PROGRAM PrgMqttCom_Blinds_Publisher
VAR
	fbMqttClient : FB_IotMqttClient;
	bSetParameter : BOOL := TRUE;
	bConnect : BOOL := TRUE;
	
	(* published message *)
	sTopicSelectRoom : STRING(255);//:= 'Staff Room';
	sTopicSelectBulkCommand : STRING(255) := 'Blind Selection';
	//sTopicSelectBoardroom : STRING(255) := 'Boardroom';
	
	bSelectStaffRoom : BOOL;
	bSelectCommunalArea : BOOL;
	bSelectBoardroom : BOOL;
	
	sPayloadCommand : STRING(255);// := 'Up';
//	sPayloadCommandDown : STRING(255) := 'Down';
//	sPayloadCommandStop : STRING(255) := 'Stop';
//	sPayloadCommandTilt : STRING(255) := 'Tilt';

	bCommandUp : BOOL;
	bCommandDown : BOOL;
	bCommandStop : BOOL;
	bCommandTilt : BOOL;
	
	bulkCommandPackage :STRING;
	
	i: INT;
	fbTimer : TON := (PT:=T#1S);
	fbTimerTilt : TON := (PT:=T#0.5S);
	
	fbMessageQueue : FB_IotMqttMessageQueue;
	fbMessage : FB_IotMqttMessage;
	
	hrErrorOccurred : HRESULT; // contains the latest occurred error
END_VAR

IF bSetParameter THEN
	bSetParameter := FALSE;
	fbMqttClient.sHostName:= '10.199.143.2';
	fbMqttClient.nHostPort:= 1883;
	fbMqttClient.sClientId:= 'CX2040_Blinds'; 
	fbMqttClient.sTopicPrefix:= ''; 
	fbMqttClient.nKeepAlive:= 60; 
//	fbMqttClient.sUserName:= ;
//	fbMqttClient.sUserPassword:= ; 
//	fbMqttClient.stWill:= ; 
//	fbMqttClient.stTLS:= ;
	fbMqttClient.ipMessageQueue := fbMessageQueue;
END_IF

fbMqttClient.Execute(bConnect);
IF fbMqttClient.bError THEN
	// add your error logging here
	hrErrorOccurred := fbMqttClient.hrErrorCode;
END_IF

IF bSelectStaffRoom THEN
	bSelectStaffRoom := FALSE;
	sTopicSelectRoom := 'Staff Room';
	bulkCommandPackage := fConvertBoolArrayToString(boolArray := BackgroundComms.BlindCommandTable[0].SelectBlindsBulkCommand);
END_IF

IF bSelectCommunalArea THEN
	bSelectCommunalArea := FALSE;
	sTopicSelectRoom := 'Communal Area';
	bulkCommandPackage := fConvertBoolArrayToString(boolArray := BackgroundComms.BlindCommandTable[1].SelectBlindsBulkCommand);
END_IF

IF bSelectBoardroom THEN
	bSelectBoardroom := FALSE;
	sTopicSelectRoom := 'Boardroom';
	bulkCommandPackage := fConvertBoolArrayToString(boolArray := BackgroundComms.BlindCommandTable[2].SelectBlindsBulkCommand);
END_IF



IF bCommandUp THEN
	bCommandUp := FALSE;
	sPayloadCommand := 'Up';
	IF sTopicSelectRoom = 'Staff Room' THEN
		bSelectStaffRoom := TRUE;
	ELSIF sTopicSelectRoom = 'Communal Area' THEN
		bulkCommandPackage := fConvertBoolArrayToString(boolArray := BackgroundComms.BlindCommandTable[1].SelectBlindsBulkCommand);
	ELSIF sTopicSelectRoom = 'Boardroom' THEN
		bulkCommandPackage := fConvertBoolArrayToString(boolArray := BackgroundComms.BlindCommandTable[2].SelectBlindsBulkCommand);
	END_IF
END_IF

IF bCommandDown THEN
	bCommandDown := FALSE;
	sPayloadCommand := 'Down';
	IF sTopicSelectRoom = 'Staff Room' THEN
		bSelectStaffRoom := TRUE;//bulkCommandPackage := fConvertBoolArrayToString(boolArray := BackgroundComms.BlindCommandTable[0].SelectBlindsBulkCommand);
	ELSIF sTopicSelectRoom = 'Communal Area' THEN
		bulkCommandPackage := fConvertBoolArrayToString(boolArray := BackgroundComms.BlindCommandTable[1].SelectBlindsBulkCommand);
	ELSIF sTopicSelectRoom = 'Boardroom' THEN
		bulkCommandPackage := fConvertBoolArrayToString(boolArray := BackgroundComms.BlindCommandTable[2].SelectBlindsBulkCommand);
	END_IF
END_IF

IF bCommandStop THEN
	bCommandStop := FALSE;
	sPayloadCommand := 'Stop';
	IF sTopicSelectRoom = 'Staff Room' THEN
		bSelectStaffRoom := TRUE;//bulkCommandPackage := fConvertBoolArrayToString(boolArray := BackgroundComms.BlindCommandTable[0].SelectBlindsBulkCommand);
	ELSIF sTopicSelectRoom = 'Communal Area' THEN
		bulkCommandPackage := fConvertBoolArrayToString(boolArray := BackgroundComms.BlindCommandTable[1].SelectBlindsBulkCommand);
	ELSIF sTopicSelectRoom = 'Boardroom' THEN
		bulkCommandPackage := fConvertBoolArrayToString(boolArray := BackgroundComms.BlindCommandTable[2].SelectBlindsBulkCommand);
	END_IF
END_IF

IF bCommandTilt THEN
	bCommandTilt := FALSE;
	sPayloadCommand := 'Tilt';
	IF sTopicSelectRoom = 'Staff Room' THEN
		bSelectStaffRoom := TRUE;//bulkCommandPackage := fConvertBoolArrayToString(boolArray := BackgroundComms.BlindCommandTable[0].SelectBlindsBulkCommand);
	ELSIF sTopicSelectRoom = 'Communal Area' THEN
		bulkCommandPackage := fConvertBoolArrayToString(boolArray := BackgroundComms.BlindCommandTable[1].SelectBlindsBulkCommand);
	ELSIF sTopicSelectRoom = 'Boardroom' THEN
		bulkCommandPackage := fConvertBoolArrayToString(boolArray := BackgroundComms.BlindCommandTable[2].SelectBlindsBulkCommand);
	END_IF
END_IF





IF fbMqttClient.bConnected THEN
	IF sPayloadCommand = 'Tilt' THEN
		fbTimerTilt(IN:=TRUE);
		fbMqttClient.Publish(	sTopic:= sTopicSelectBulkCommand, 
									pPayload:= ADR(bulkCommandPackage), nPayloadSize:= LEN2(ADR(bulkCommandPackage))+1, 
									eQoS:= TcIotMqttQos.AtMostOnceDelivery, bRetain:= FALSE, bQueue:= FALSE );
		fbMqttClient.Publish(	sTopic:= sTopicSelectRoom, 
									pPayload:= ADR(sPayloadCommand), nPayloadSize:= LEN2(ADR(sPayloadCommand))+1, 
									eQoS:= TcIotMqttQos.AtMostOnceDelivery, bRetain:= FALSE, bQueue:= FALSE );
		
		IF fbTimerTilt.Q THEN // publish new payload every second
			sPayloadCommand := 'Stop';
			fbTimerTilt(IN:=FALSE);
			fbMqttClient.Publish(	sTopic:= sTopicSelectBulkCommand, 
									pPayload:= ADR(bulkCommandPackage), nPayloadSize:= LEN2(ADR(bulkCommandPackage))+1, 
									eQoS:= TcIotMqttQos.AtMostOnceDelivery, bRetain:= FALSE, bQueue:= FALSE );
			fbMqttClient.Publish(	sTopic:= sTopicSelectRoom, 
									pPayload:= ADR(sPayloadCommand), nPayloadSize:= LEN2(ADR(sPayloadCommand))+1, 
									eQoS:= TcIotMqttQos.AtMostOnceDelivery, bRetain:= FALSE, bQueue:= FALSE );			
			IF fbMqttClient.bError THEN
				// add your error logging here
				hrErrorOccurred := fbMqttClient.hrErrorCode;
			END_IF
		END_IF
	ELSE
		fbTimer(IN:=TRUE);
		IF fbTimer.Q THEN // publish new payload every second
			fbTimer(IN:=FALSE);
			fbMqttClient.Publish(	sTopic:= sTopicSelectBulkCommand, 
									pPayload:= ADR(bulkCommandPackage), nPayloadSize:= LEN2(ADR(bulkCommandPackage))+1, 
									eQoS:= TcIotMqttQos.AtMostOnceDelivery, bRetain:= FALSE, bQueue:= FALSE );
									
			fbMqttClient.Publish(	sTopic:= sTopicSelectRoom, 
									pPayload:= ADR(sPayloadCommand), nPayloadSize:= LEN2(ADR(sPayloadCommand))+1, 
									eQoS:= TcIotMqttQos.AtMostOnceDelivery, bRetain:= FALSE, bQueue:= FALSE );
			IF fbMqttClient.bError THEN
				// add your error logging here
				hrErrorOccurred := fbMqttClient.hrErrorCode;
			END_IF
		END_IF
	END_IF
END_IF

fbTimerTilt();

END_PROGRAM

(* stored: Version 1.1.0.1, ProductVersion 3.1.4024.12
   POU PrgMqttCom_Blinds_Publisher: Id {3671603f-ce1a-4877-9351-391aaefe0379}, SpecialFunc None *)
